(* CODESYS project bibliothek.library
   Company: Viessmann
   Title: GWP_Libary_Visu_1
   Placeholder: GWP_Libary_Visu_1
   Version: 0.0.1

Project tree, tasks and I/O mapping:
  libraries: GWP Library, 17.9.1 (Viessmann); Tc2_Standard, * (Beckhoff Automation GmbH); Tc2_System, * (Beckhoff Automation GmbH); Tc2_Utilities, * (Beckhoff Automation GmbH); Tc3_Module, * (Beckhoff Automation GmbH); VisuDialogs, * (System)
  DUTs/
    GVLs/
      global variables Globale_Uhr
  POUs/
    Funktionsblock/
    program MAIN [ST]
    program test [FBD]
  Version/
    global variables Global_Version
  VISUs/
    Alarmliste/
      visualisation Alarmliste
    Anlageseite_6/
      visualisation Kaeltekreis6_1
      visualisation Sollwertaenderung_C_6_3
      visualisation Zustandsanzeige
    Hauptmenu_3/
      visualisation Fusszeile_50
      visualisation Hauptmenu
      visualisation Kachel_IBN
      visualisation Kachel_Konfiguration
      visualisation Kachel_Kontakt
      visualisation Kachel_Login
      visualisation Kachel_Sollwerte
      visualisation Kachel_Sprachen
      visualisation Kachel_Uhrzeit_einstellen
      visualisation Kachel_Verlaufsdiagramm
      visualisation Kontaktseite
      visualisation Uhr_einstellen
    Heizkurven/
      visualisation Heizkurve
    Home/
      visualisation Auswahlmenue
      visualisation Ein_Aus_Schalter
      visualisation Home_Standard_50
      visualisation RI_Schema_50
    IBN/
      visualisation IO_Auswahl
      visualisation Liste_AI
      visualisation Liste_AO
      visualisation Liste_DI
      visualisation Liste_DO
      visualisation SW_IBN_Einstellungen_K
    Infoseite/
      visualisation Infoliste
      visualisation Infoseite
    Sollwertmenu_9/
      Sollwerte Einstellungen/
        visualisation SW_Einstellungen_C
        visualisation SW_Einstellungen_Faktor
        visualisation SW_Einstellungen_K
        visualisation SW_Einstellungen_min
        visualisation SW_Einstellungen_ms
        visualisation SW_zuruecksetzen
      Sollwertmenu/
        visualisation Sollwertmenu
      Wärmegewinnung/
        UWP/
          visualisation SW_WG_UWP_Verd
          visualisation SW_WG_UWP_Verd_Liste
        visualisation Kachel_Abtauspeicher
        visualisation Kachel_Abtauungen
        visualisation Kachel_Abwaerme
        visualisation Kachel_Erdsonden
        visualisation Kachel_Grundwasser
        visualisation Kachel_Luft
        visualisation Kachel_Tiefhaltung
        visualisation Kachel_UWP_Verd
        visualisation Sollwertmenu_Waermegewinnung
      Wärmepumpe/
        EEV/
          visualisation SW_WP_EEV
          visualisation SW_WP_EEV_Liste
        Einsatzgrenzen/
          visualisation SW_WP_Einsatzgrenzen
          visualisation SW_WP_Einsatzgrenzen_Liste
        visualisation Kachel_Allgemein
        visualisation Kachel_EEV
        visualisation Kachel_Einsatzgrenzen
        visualisation Kachel_Verdichter
        visualisation Sollwertmenu_Waermepumpe
      Wärmesenke/
        visualisation Kachel_Heizgruppen
        visualisation Kachel_Hochhaltung
        visualisation Kachel_HWP
        visualisation Kachel_TWW
        visualisation Kachel_UWP_Verfl
        visualisation Sollwertmenu_Waermesenke
    Sprache/
      visualisation Spracheistellungen
    Zeitprogramm/
      visualisation EIn_Aus_Zeit_aendern
      visualisation Wochenuhr_W7
      visualisation Wochenuhr_W7_Liste
    image pool Icon
    text list Sprachen
    visualisation test_1
  00000000-0000-0000-0000-000000000000|C:\Users\kuzr\Documents\Visual Studio 2013\Bildersammlung_VI\IC_102000\energietraeger_biomasse_fehler.png
  00000000-0000-0000-0000-000000000000|C:\Users\kuzr\Documents\Visual Studio 2013\Bildersammlung_VI\IC_102000\energietraeger_biomasse_inaktiv.png
  00000000-0000-0000-0000-000000000000|C:\Users\kuzr\Documents\Visual Studio 2013\Bildersammlung_VI\IC_102000\energietraeger_gas.png
  00000000-0000-0000-0000-000000000000|C:\Users\kuzr\Documents\Visual Studio 2013\Bildersammlung_VI\IC_102000\energietraeger_gas_fehler.png
  00000000-0000-0000-0000-000000000000|C:\Users\kuzr\Documents\Visual Studio 2013\Bildersammlung_VI\IC_102000\energietraeger_naturwaerme.png
  00000000-0000-0000-0000-000000000000|C:\Users\kuzr\Documents\Visual Studio 2013\Bildersammlung_VI\IC_102000\energietraeger_naturwaerme_fehler (2).png
  00000000-0000-0000-0000-000000000000|C:\Users\kuzr\Documents\Visual Studio 2013\Bildersammlung_VI\IC_102000\energietraeger_naturwaerme_fehler.png
  00000000-0000-0000-0000-000000000000|C:\Users\kuzr\Documents\Visual Studio 2013\Bildersammlung_VI\IC_102000\energietraeger_naturwaerme_inaktiv.png
  00000000-0000-0000-0000-000000000000|C:\Users\kuzr\Documents\Visual Studio 2013\Bildersammlung_VI\IC_102000\energietraeger_oel.png
  00000000-0000-0000-0000-000000000000|C:\Users\kuzr\Documents\Visual Studio 2013\Bildersammlung_VI\IC_102000\energietraeger_oel_inaktiv.png
  00000000-0000-0000-0000-000000000000|C:\Users\kuzr\Documents\Visual Studio 2013\Bildersammlung_VI\IC_102000\heizkreis_direkt (2).png
  00000000-0000-0000-0000-000000000000|C:\Users\kuzr\Documents\Visual Studio 2013\Bildersammlung_VI\IC_102000\heizkreis_direkt.png
  00000000-0000-0000-0000-000000000000|C:\Users\kuzr\Documents\Visual Studio 2013\Bildersammlung_VI\IC_102000\heizkreis_direkt_fehler.png
  00000000-0000-0000-0000-000000000000|C:\Users\kuzr\Documents\Visual Studio 2013\Bildersammlung_VI\IC_102000\heizkreis_direkt_inaktiv (2).png
  00000000-0000-0000-0000-000000000000|C:\Users\kuzr\Documents\Visual Studio 2013\Bildersammlung_VI\IC_102000\heizkreis_direkt_inaktiv.png
  00000000-0000-0000-0000-000000000000|C:\Users\kuzr\Documents\Visual Studio 2013\Bildersammlung_VI\IC_102000\heizkreis_fussbodenheizung.png
  00000000-0000-0000-0000-000000000000|C:\Users\kuzr\Documents\Visual Studio 2013\Bildersammlung_VI\IC_102000\heizkreis_fussbodenheizung_fehler.png
  00000000-0000-0000-0000-000000000000|C:\Users\kuzr\Documents\Visual Studio 2013\Bildersammlung_VI\IC_102000\heizkreis_fussbodenheizung_inaktiv.png
  00000000-0000-0000-0000-000000000000|C:\Users\kuzr\Documents\Visual Studio 2013\Bildersammlung_VI\IC_102000\heizkreis_mischer.png
  00000000-0000-0000-0000-000000000000|C:\Users\kuzr\Documents\Visual Studio 2013\Bildersammlung_VI\IC_102000\heizkreis_mischer_fehler.png
  00000000-0000-0000-0000-000000000000|C:\Users\kuzr\Documents\Visual Studio 2013\Bildersammlung_VI\IC_102000\heizkreis_mischer_inaktiv.png
  00000000-0000-0000-0000-000000000000|C:\Users\kuzr\Documents\Visual Studio 2013\Bildersammlung_VI\IC_102000\IC_102015_klappen_02.png
  00000000-0000-0000-0000-000000000000|C:\Users\kuzr\Documents\Visual Studio 2013\Bildersammlung_VI\IC_102000\klappen_01 (2).png
  00000000-0000-0000-0000-000000000000|C:\Users\kuzr\Documents\Visual Studio 2013\Bildersammlung_VI\IC_102000\klappen_01.png
  00000000-0000-0000-0000-000000000000|C:\Users\kuzr\Documents\Visual Studio 2013\Bildersammlung_VI\IC_102000\klappen_02.png
  00000000-0000-0000-0000-000000000000|C:\Users\kuzr\Documents\Visual Studio 2013\Bildersammlung_VI\IC_102000\komponente_detail_heizkreis.png
  00000000-0000-0000-0000-000000000000|C:\Users\kuzr\Documents\Visual Studio 2013\Bildersammlung_VI\IC_102000\komponente_detail_klappe (2).png
  00000000-0000-0000-0000-000000000000|C:\Users\kuzr\Documents\Visual Studio 2013\Bildersammlung_VI\IC_102000\komponente_detail_klappe.png
  00000000-0000-0000-0000-000000000000|C:\Users\kuzr\Documents\Visual Studio 2013\Bildersammlung_VI\IC_102000\komponente_detail_klappe_fehler (2).png
  00000000-0000-0000-0000-000000000000|C:\Users\kuzr\Documents\Visual Studio 2013\Bildersammlung_VI\IC_102000\komponente_detail_klappe_fehler.png
  00000000-0000-0000-0000-000000000000|C:\Users\kuzr\Documents\Visual Studio 2013\Bildersammlung_VI\IC_102000\komponente_detail_klappe_inaktiv.png
  00000000-0000-0000-0000-000000000000|C:\Users\kuzr\Documents\Visual Studio 2013\Bildersammlung_VI\IC_102000\komponente_detail_klappe_inaktiv_2.png
  00000000-0000-0000-0000-000000000000|C:\Users\kuzr\Documents\Visual Studio 2013\Bildersammlung_VI\IC_102000\komponente_detail_mischer_01.png
  00000000-0000-0000-0000-000000000000|C:\Users\kuzr\Documents\Visual Studio 2013\Bildersammlung_VI\IC_102000\komponente_detail_mischer_02.png
  00000000-0000-0000-0000-000000000000|C:\Users\kuzr\Documents\Visual Studio 2013\Bildersammlung_VI\IC_102000\komponente_detail_mischer_fehler.png
  00000000-0000-0000-0000-000000000000|C:\Users\kuzr\Documents\Visual Studio 2013\Bildersammlung_VI\IC_102000\komponente_detail_mischer_inaktiv.png
  00000000-0000-0000-0000-000000000000|C:\Users\kuzr\Documents\Visual Studio 2013\Bildersammlung_VI\IC_102000\komponente_detail_pumpe.png
  00000000-0000-0000-0000-000000000000|C:\Users\kuzr\Documents\Visual Studio 2013\Bildersammlung_VI\IC_102000\komponente_detail_pumpe_fehler.png
  00000000-0000-0000-0000-000000000000|C:\Users\kuzr\Documents\Visual Studio 2013\Bildersammlung_VI\IC_102000\komponente_detail_pumpe_inaktiv.png
  00000000-0000-0000-0000-000000000000|C:\Users\kuzr\Documents\Visual Studio 2013\Bildersammlung_VI\IC_102000\mischer_01.png
  00000000-0000-0000-0000-000000000000|C:\Users\kuzr\Documents\Visual Studio 2013\Bildersammlung_VI\IC_102000\mischer_02.png
  00000000-0000-0000-0000-000000000000|C:\Users\kuzr\Documents\Visual Studio 2013\Bildersammlung_VI\IC_102000\mischer_03.png
  00000000-0000-0000-0000-000000000000|C:\Users\kuzr\Documents\Visual Studio 2013\Bildersammlung_VI\IC_102000\mischer_04.png
  00000000-0000-0000-0000-000000000000|C:\Users\kuzr\Documents\Visual Studio 2013\Bildersammlung_VI\IC_102000\mischer_05.png
  00000000-0000-0000-0000-000000000000|C:\Users\kuzr\Documents\Visual Studio 2013\Bildersammlung_VI\IC_102000\mischer_06.png
  00000000-0000-0000-0000-000000000000|C:\Users\kuzr\Documents\Visual Studio 2013\Bildersammlung_VI\IC_102000\mischer_07.png
  00000000-0000-0000-0000-000000000000|C:\Users\kuzr\Documents\Visual Studio 2013\Bildersammlung_VI\IC_102000\mischer_08.png
  00000000-0000-0000-0000-000000000000|C:\Users\kuzr\Documents\Visual Studio 2013\Bildersammlung_VI\IC_102000\mischer_09.png
  00000000-0000-0000-0000-000000000000|C:\Users\kuzr\Documents\Visual Studio 2013\Bildersammlung_VI\IC_102000\mischer_10.png
  00000000-0000-0000-0000-000000000000|C:\Users\kuzr\Documents\Visual Studio 2013\Bildersammlung_VI\IC_102000\mischer_11.png
  00000000-0000-0000-0000-000000000000|C:\Users\kuzr\Documents\Visual Studio 2013\Bildersammlung_VI\IC_102000\mischer_12.png
  00000000-0000-0000-0000-000000000000|C:\Users\kuzr\Documents\Visual Studio 2013\Bildersammlung_VI\IC_102000\pumpe_links.png
  00000000-0000-0000-0000-000000000000|C:\Users\kuzr\Documents\Visual Studio 2013\Bildersammlung_VI\IC_102000\pumpe_oben.png
  00000000-0000-0000-0000-000000000000|C:\Users\kuzr\Documents\Visual Studio 2013\Bildersammlung_VI\IC_102000\pumpe_rechts.png
  00000000-0000-0000-0000-000000000000|C:\Users\kuzr\Documents\Visual Studio 2013\Bildersammlung_VI\IC_102000\pumpe_unten.png
  00000000-0000-0000-0000-000000000000|C:\Users\kuzr\Documents\Visual Studio 2013\Bildersammlung_VI\IC_102000\speicher_eis.png
  00000000-0000-0000-0000-000000000000|C:\Users\kuzr\Documents\Visual Studio 2013\Bildersammlung_VI\IC_102000\speicher_eis_fehler.png
  00000000-0000-0000-0000-000000000000|C:\Users\kuzr\Documents\Visual Studio 2013\Bildersammlung_VI\IC_102000\speicher_eis_inaktiv.png
  00000000-0000-0000-0000-000000000000|C:\Users\kuzr\Documents\Visual Studio 2013\Bildersammlung_VI\IC_102000\speicher_heizen.png
  00000000-0000-0000-0000-000000000000|C:\Users\kuzr\Documents\Visual Studio 2013\Bildersammlung_VI\IC_102000\speicher_heizen_fehler.png
  00000000-0000-0000-0000-000000000000|C:\Users\kuzr\Documents\Visual Studio 2013\Bildersammlung_VI\IC_102000\speicher_heizen_inaktiv.png
  00000000-0000-0000-0000-000000000000|C:\Users\kuzr\Documents\Visual Studio 2013\Bildersammlung_VI\IC_102000\speicher_warmwasser.png
  00000000-0000-0000-0000-000000000000|C:\Users\kuzr\Documents\Visual Studio 2013\Bildersammlung_VI\IC_102000\speicher_warmwasser_fehler.png
  00000000-0000-0000-0000-000000000000|C:\Users\kuzr\Documents\Visual Studio 2013\Bildersammlung_VI\IC_102000\speicher_warmwasser_inaktiv.png
  00000000-0000-0000-0000-000000000000|C:\Users\kuzr\Documents\Visual Studio 2013\Bildersammlung_VI\IC_102000\energietraeger_biomasse.png
  00000000-0000-0000-0000-000000000000|C:\Users\kuzr\Documents\Visual Studio 2013\Bildersammlung_VI\IC_106000\komponente_brenner.png
  00000000-0000-0000-0000-000000000000|C:\Users\kuzr\Documents\Visual Studio 2013\Bildersammlung_VI\IC_106000\komponente_brenner_fehler.png
  00000000-0000-0000-0000-000000000000|C:\Users\kuzr\Documents\Visual Studio 2013\Bildersammlung_VI\IC_106000\komponente_brenner_inaktiv.png
  00000000-0000-0000-0000-000000000000|C:\Users\kuzr\Documents\Visual Studio 2013\Bildersammlung_VI\IC_106000\speicher.png
  00000000-0000-0000-0000-000000000000|C:\Users\kuzr\Documents\Visual Studio 2013\Bildersammlung_VI\IC_106000\speicher_eis.png
  00000000-0000-0000-0000-000000000000|C:\Users\kuzr\Documents\Visual Studio 2013\Bildersammlung_VI\IC_106000\system_leistung_nicht_touchbar.png
  00000000-0000-0000-0000-000000000000|C:\Users\kuzr\Documents\Visual Studio 2013\Bildersammlung_VI\IC_106000\system_leistung_touchbar.png
  00000000-0000-0000-0000-000000000000|C:\Users\kuzr\Documents\Visual Studio 2013\Bildersammlung_VI\IC_106000\waermetauscher.png
  00000000-0000-0000-0000-000000000000|C:\Users\kuzr\Documents\Visual Studio 2013\Bildersammlung_VI\IC_106000\weiche.png
  00000000-0000-0000-0000-000000000000|C:\Users\kuzr\Documents\Visual Studio 2013\Bildersammlung_VI\IC_108000\komponente_brenner_fehler.png
  00000000-0000-0000-0000-000000000000|C:\Users\kuzr\Documents\Visual Studio 2013\Bildersammlung_VI\IC_108000\komponente_brenner_inaktiv.png
  00000000-0000-0000-0000-000000000000|C:\Users\kuzr\Documents\Visual Studio 2013\Bildersammlung_VI\IC_108000\speicher.png
  00000000-0000-0000-0000-000000000000|C:\Users\kuzr\Documents\Visual Studio 2013\Bildersammlung_VI\IC_108000\speicher_eis.png
  00000000-0000-0000-0000-000000000000|C:\Users\kuzr\Documents\Visual Studio 2013\Bildersammlung_VI\IC_108000\komponente_brenner.png
  00000000-0000-0000-0000-000000000000|C:\Users\kuzr\Documents\Visual Studio 2013\Bildersammlung_VI\IC_111000\bildschirm_reinigen.png
  00000000-0000-0000-0000-000000000000|C:\Users\kuzr\Documents\Visual Studio 2013\Bildersammlung_VI\IC_111000\dokumentation.png
  00000000-0000-0000-0000-000000000000|C:\Users\kuzr\Documents\Visual Studio 2013\Bildersammlung_VI\IC_111000\kontaktdaten_nutzer.png
  00000000-0000-0000-0000-000000000000|C:\Users\kuzr\Documents\Visual Studio 2013\Bildersammlung_VI\IC_111000\kontaktdaten_viessmann.png
  00000000-0000-0000-0000-000000000000|C:\Users\kuzr\Documents\Visual Studio 2013\Bildersammlung_VI\IC_111000\nutzeranmeldung.png
  00000000-0000-0000-0000-000000000000|C:\Users\kuzr\Documents\Visual Studio 2013\Bildersammlung_VI\IC_111000\oberflaeche_schließen.png
  00000000-0000-0000-0000-000000000000|C:\Users\kuzr\Documents\Visual Studio 2013\Bildersammlung_VI\IC_111000\pruefbetrieb.png
  00000000-0000-0000-0000-000000000000|C:\Users\kuzr\Documents\Visual Studio 2013\Bildersammlung_VI\IC_111000\system_konfigurieren.png
  00000000-0000-0000-0000-000000000000|C:\Users\kuzr\Documents\Visual Studio 2013\Bildersammlung_VI\IC_111000\betriebszaehler_zuruecksetzen.png
  00000000-0000-0000-0000-000000000000|C:\Users\kuzr\Documents\Visual Studio 2013\Bildersammlung_VI\IC_112000\abschaltbetrieb.png
  00000000-0000-0000-0000-000000000000|C:\Users\kuzr\Documents\Visual Studio 2013\Bildersammlung_VI\IC_112000\aktiv.png
  00000000-0000-0000-0000-000000000000|C:\Users\kuzr\Documents\Visual Studio 2013\Bildersammlung_VI\IC_112000\an.png
  00000000-0000-0000-0000-000000000000|C:\Users\kuzr\Documents\Visual Studio 2013\Bildersammlung_VI\IC_112000\astatur_01.png
  00000000-0000-0000-0000-000000000000|C:\Users\kuzr\Documents\Visual Studio 2013\Bildersammlung_VI\IC_112000\auf.png
  00000000-0000-0000-0000-000000000000|C:\Users\kuzr\Documents\Visual Studio 2013\Bildersammlung_VI\IC_112000\aus.png
  00000000-0000-0000-0000-000000000000|C:\Users\kuzr\Documents\Visual Studio 2013\Bildersammlung_VI\IC_112000\bedingung_erfuellt.png
  00000000-0000-0000-0000-000000000000|C:\Users\kuzr\Documents\Visual Studio 2013\Bildersammlung_VI\IC_112000\bedingung_nicht_erfuellt.png
  00000000-0000-0000-0000-000000000000|C:\Users\kuzr\Documents\Visual Studio 2013\Bildersammlung_VI\IC_112000\email_prueftaste.png
  00000000-0000-0000-0000-000000000000|C:\Users\kuzr\Documents\Visual Studio 2013\Bildersammlung_VI\IC_112000\erfuellt.png
  00000000-0000-0000-0000-000000000000|C:\Users\kuzr\Documents\Visual Studio 2013\Bildersammlung_VI\IC_112000\exportieren.png
  00000000-0000-0000-0000-000000000000|C:\Users\kuzr\Documents\Visual Studio 2013\Bildersammlung_VI\IC_112000\frostschutzbetrieb.png
  00000000-0000-0000-0000-000000000000|C:\Users\kuzr\Documents\Visual Studio 2013\Bildersammlung_VI\IC_112000\haeckchen_ungesetzt (2).png
  00000000-0000-0000-0000-000000000000|C:\Users\kuzr\Documents\Visual Studio 2013\Bildersammlung_VI\IC_112000\haeckchen_ungesetzt.png
  00000000-0000-0000-0000-000000000000|C:\Users\kuzr\Documents\Visual Studio 2013\Bildersammlung_VI\IC_112000\home.png
  00000000-0000-0000-0000-000000000000|C:\Users\kuzr\Documents\Visual Studio 2013\Bildersammlung_VI\IC_112000\home_uebersicht.png
  00000000-0000-0000-0000-000000000000|C:\Users\kuzr\Documents\Visual Studio 2013\Bildersammlung_VI\IC_112000\inaktiv.png
  00000000-0000-0000-0000-000000000000|C:\Users\kuzr\Documents\Visual Studio 2013\Bildersammlung_VI\IC_112000\intervall.png
  00000000-0000-0000-0000-000000000000|C:\Users\kuzr\Documents\Visual Studio 2013\Bildersammlung_VI\IC_112000\Itastatur_03.png
  00000000-0000-0000-0000-000000000000|C:\Users\kuzr\Documents\Visual Studio 2013\Bildersammlung_VI\IC_112000\ja.png
  00000000-0000-0000-0000-000000000000|C:\Users\kuzr\Documents\Visual Studio 2013\Bildersammlung_VI\IC_112000\kopieren.png
  00000000-0000-0000-0000-000000000000|C:\Users\kuzr\Documents\Visual Studio 2013\Bildersammlung_VI\IC_112000\laden.png
  00000000-0000-0000-0000-000000000000|C:\Users\kuzr\Documents\Visual Studio 2013\Bildersammlung_VI\IC_112000\listenansicht.png
  00000000-0000-0000-0000-000000000000|C:\Users\kuzr\Documents\Visual Studio 2013\Bildersammlung_VI\IC_112000\meldelisten_archiv.png
  00000000-0000-0000-0000-000000000000|C:\Users\kuzr\Documents\Visual Studio 2013\Bildersammlung_VI\IC_112000\meldelisten_einstellungen.png
  00000000-0000-0000-0000-000000000000|C:\Users\kuzr\Documents\Visual Studio 2013\Bildersammlung_VI\IC_112000\meldungen_weiterleiten.png
  00000000-0000-0000-0000-000000000000|C:\Users\kuzr\Documents\Visual Studio 2013\Bildersammlung_VI\IC_112000\menue.png
  00000000-0000-0000-0000-000000000000|C:\Users\kuzr\Documents\Visual Studio 2013\Bildersammlung_VI\IC_112000\minus.png
  00000000-0000-0000-0000-000000000000|C:\Users\kuzr\Documents\Visual Studio 2013\Bildersammlung_VI\IC_112000\nein.png
  00000000-0000-0000-0000-000000000000|C:\Users\kuzr\Documents\Visual Studio 2013\Bildersammlung_VI\IC_112000\nicht_erfuellt.png
  00000000-0000-0000-0000-000000000000|C:\Users\kuzr\Documents\Visual Studio 2013\Bildersammlung_VI\IC_112000\normalbetrieb.png
  00000000-0000-0000-0000-000000000000|C:\Users\kuzr\Documents\Visual Studio 2013\Bildersammlung_VI\IC_112000\pfeil_rechts.png
  00000000-0000-0000-0000-000000000000|C:\Users\kuzr\Documents\Visual Studio 2013\Bildersammlung_VI\IC_112000\plus.png
  00000000-0000-0000-0000-000000000000|C:\Users\kuzr\Documents\Visual Studio 2013\Bildersammlung_VI\IC_112000\quittieren_aus.png
  00000000-0000-0000-0000-000000000000|C:\Users\kuzr\Documents\Visual Studio 2013\Bildersammlung_VI\IC_112000\quittierena_an.png
  00000000-0000-0000-0000-000000000000|C:\Users\kuzr\Documents\Visual Studio 2013\Bildersammlung_VI\IC_112000\radiobutton_gesetzt.png
  00000000-0000-0000-0000-000000000000|C:\Users\kuzr\Documents\Visual Studio 2013\Bildersammlung_VI\IC_112000\radiobutton_ungesetzt.png
  text list GlobalTextList
*)

// DUTs/GVLs/Globale_Uhr
{attribute 'qualified_only'}
VAR_GLOBAL
	
	   systemtimestruct		: timestruct;   
END_VAR

// Version/Global_Version
{attribute 'TcGenerated'}
// This function has been automatically generated from the project information.
VAR_GLOBAL CONSTANT
	{attribute 'const_non_replaced'}
	{attribute 'linkalways'}
	stLibVersion_GWP_Libary_Visu_1 : ST_LibVersion := (iMajor := 0, iMinor := 0, iBuild := 1, iRevision := 0, sVersion := '0.0.1');
END_VAR

// POUs/MAIN
PROGRAM MAIN
VAR

	

END_VAR

END_PROGRAM

// POUs/test
PROGRAM test
VAR

	
	Globale_Zeit_0: Globale_Zeit;
    CLK_W_0: CLK_W;
	
	GR_2_0: GR_2;
	
	


	
	Logger_0: Logger;
	GR_4_mit_RE_0: GR_4_mit_RE;
	CLK_W7_0: CLK_W7;
END_VAR

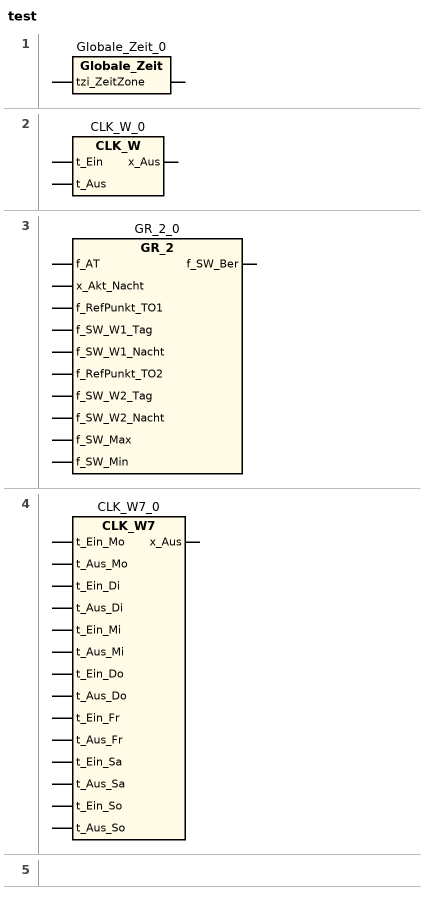
// NETWORK 1
Globale_Zeit_0(); // Globale_Zeit

// NETWORK 2
CLK_W_0(); // CLK_W

// NETWORK 3
GR_2_0(); // GR_2

// NETWORK 4
CLK_W7_0(); // CLK_W7

// NETWORK 5

END_PROGRAM

// VISUs/Alarmliste/Alarmliste
VISUALIZATION Alarmliste  // 800x430
END_VISUALIZATION

// VISUs/Anlageseite_6/Kaeltekreis6_1
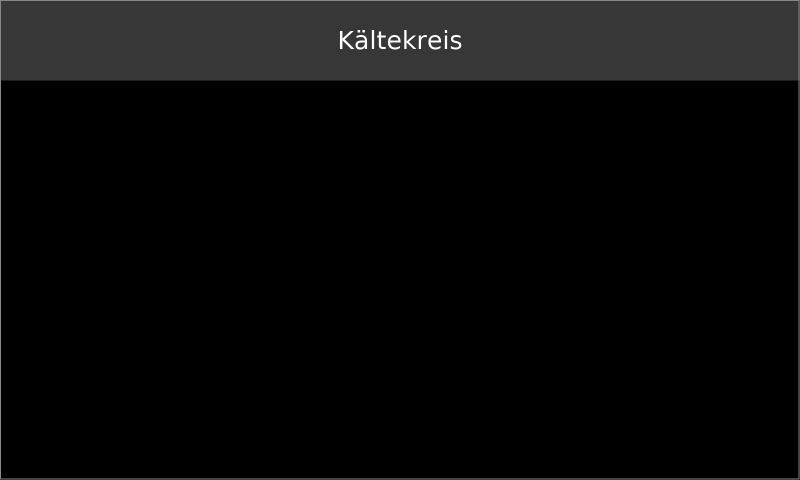
VISUALIZATION Kaeltekreis6_1  // 800x480
    Rectangle (0,0 800x80), "Kältekreis"
END_VISUALIZATION

// VISUs/Anlageseite_6/Sollwertaenderung_C_6_3
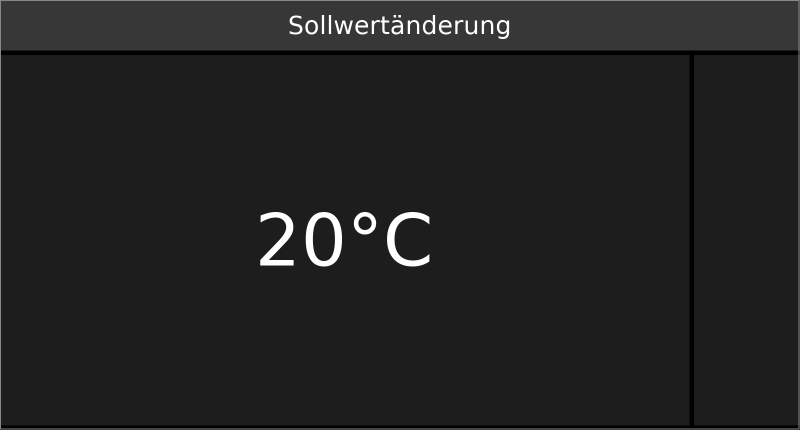
VISUALIZATION Sollwertaenderung_C_6_3  // 800x430
    Rectangle (0,0 800x50), "Sollwertänderung"
    Rectangle (0,55 689x370), "20°C"
    Rectangle (694,55 106x370)
END_VISUALIZATION

// VISUs/Anlageseite_6/Zustandsanzeige
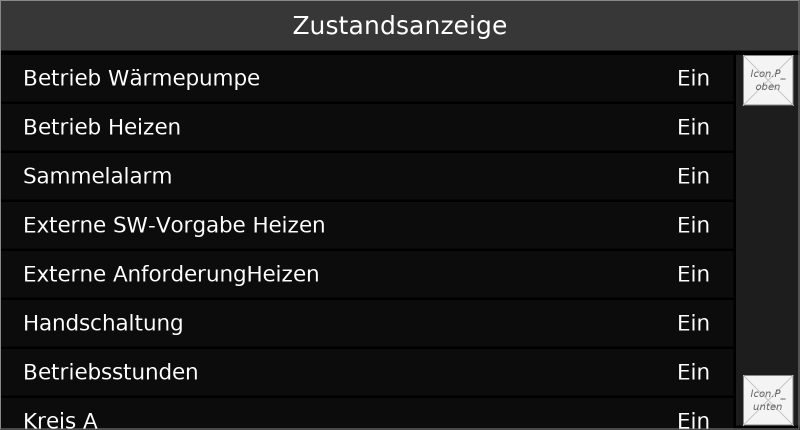
VISUALIZATION Zustandsanzeige  // 800x430
VAR_IN_OUT
	auf:BOOL;
		
END_VAR
    Image (1113,281 30x116), image: Icon.waermetauscher
    Group (0,0 800x640)
        Rectangle (0,0 800x50), "Zustandsanzeige"
        Group (0,430 800x50)
            Rectangle (0,0 800x50)
            Image (25,0 50x50), image: Icon.home
            Image (425,0 50x50), image: Icon.reinnavigieren
            Image (625,0 50x50), image: Icon.warnung_rot
            Image (125,0 50x50), image: Icon.zurueck
            Image (325,0 50x50), image: Icon.reinnavigieren
            Image (325,0 50x50), image: Icon.p_links
            Image (425,0 50x50), image: Icon.P_rechts
        Rectangle (0,55 733x46)
        Label (20,55 479x46), "Betrieb Wärmepumpe"
        Rectangle (0,104 733x46)
        Label (20,104 479x46), "Betrieb Heizen"
        Rectangle (0,153 733x46)
        Label (20,153 479x46), "Sammelalarm"
        Rectangle (0,202 733x46)
        Label (20,202 479x46), "Externe SW-Vorgabe Heizen"
        Rectangle (0,251 733x46)
        Label (20,251 479x46), "Externe AnforderungHeizen"
        Rectangle (0,300 733x46)
        Label (20,300 479x46), "Handschaltung"
        Rectangle (0,349 733x46)
        Label (20,349 479x46), "Betriebsstunden"
        Rectangle (583,55 130x46), "Ein"
        Rectangle (583,104 130x46), "Ein"
        Rectangle (0,398 733x46)
        Label (20,398 479x46), "Kreis A"
        Rectangle (0,447 733x46)
        Label (20,447 479x46), "Kreis B"
        Rectangle (0,496 733x46)
        Label (20,496 479x46), "Stufe 1"
        Rectangle (0,545 733x46)
        Label (20,545 479x46), "Stufe 2"
        Rectangle (583,545 130x46), "Ein"
        Rectangle (0,594 733x46)
        Label (20,594 479x46), "Stufe 3"
        Rectangle (583,153 130x46), "Ein"
        Rectangle (583,202 130x46), "Ein"
        Rectangle (583,251 130x46), "Ein"
        Rectangle (583,349 130x46), "Ein"
        Rectangle (583,300 130x46), "Ein"
        Rectangle (583,398 130x46), "Ein"
        Rectangle (583,447 130x46), "Ein"
        Rectangle (583,496 130x46), "Ein"
        Rectangle (583,594 130x46), "Ein"
        Rectangle (736,55 64x370)
        Image (743,55 50x50), image: Icon.P_oben
            OnMouseClick: write the text variable via Default
        Image (743,375 50x50), image: Icon.P_unten
END_VISUALIZATION

// VISUs/Hauptmenu_3/Fusszeile_50
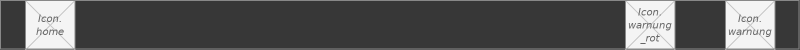
VISUALIZATION Fusszeile_50  // 800x50
    Group (0,0 800x50)
        Rectangle (0,0 800x50)
        Image (625,0 50x50), image: Icon.warnung_rot
            OnMouseClick: execute { GWP_Library.Visu.i_Frame_Index:=0; }
        Image (25,0 50x50), image: Icon.home
            OnMouseClick:  Assign=Home_Standard_50, Type=Assignment
            OnMouseClick: execute { GWP_Library.Visu.i_Frame_Index:=0; }
        Image (725,0 50x50), image: Icon.warnung
            OnMouseClick:  Assign=Infoseite, Type=Assignment
            OnMouseClick: execute { GWP_Library.Visu.i_Frame_Index:=0; }
END_VISUALIZATION

// VISUs/Hauptmenu_3/Hauptmenu
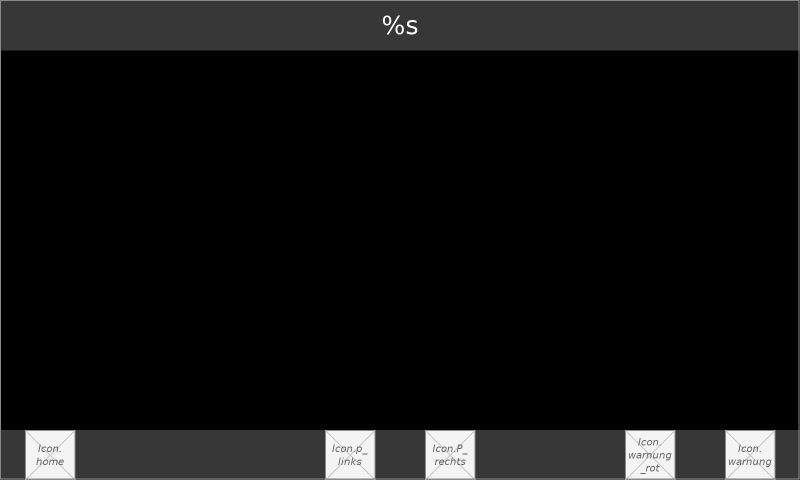
VISUALIZATION Hauptmenu  // 800x480
VAR_IN_OUT
		
END_VAR

VAR
	i_verschieben:INT;

END_VAR
    Image (425,430 50x50), image: Icon.reinnavigieren
    Image (325,430 50x50), image: Icon.reinnavigieren
    Rectangle (0,0 800x50), "%s", text list: 'Sprachen', text index: 32
    Frame (0,430 800x50)
        shows Fusszeile_50()
    Image (425,430 50x50), image: Icon.P_rechts
        OnMouseClick: execute {
            IF i_verschieben>-800 THEN
            	i_verschieben:=i_verschieben-800;
            END_IF
        }
    Image (325,430 50x50), image: Icon.p_links
        OnMouseClick: execute {
            IF i_verschieben<0 THEN
            	i_verschieben:=i_verschieben+800;
            END_IF
        }
    Rectangle (88,515 454x57), "Kachel 1: 0;55 *** Kachel 2: 201;55 *** Kachel 3: 402;55 *** Kachel 4: 604;55 Kachel 5: 0;242 *** Kachel 6: 201;242 *** Kachel 7: 402;242 *** Kachel 8: 604;242"
END_VISUALIZATION

// VISUs/Hauptmenu_3/Kachel_IBN
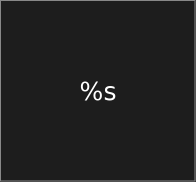
VISUALIZATION Kachel_IBN  // 196x182
    Rectangle (0,0 196x182), "%s", text list: 'Sprachen', text index: 38
END_VISUALIZATION

// VISUs/Hauptmenu_3/Kachel_Konfiguration
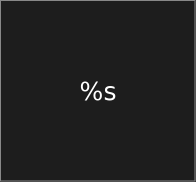
VISUALIZATION Kachel_Konfiguration  // 196x182
    Rectangle (0,0 196x182), "%s", text list: 'Sprachen', text index: 39
END_VISUALIZATION

// VISUs/Hauptmenu_3/Kachel_Kontakt
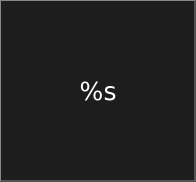
VISUALIZATION Kachel_Kontakt  // 196x182
    Rectangle (0,0 196x182), "%s", text list: 'Sprachen', text index: 40
END_VISUALIZATION

// VISUs/Hauptmenu_3/Kachel_Login
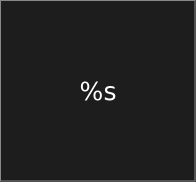
VISUALIZATION Kachel_Login  // 196x182
    Rectangle (0,0 196x182), "%s", text list: 'Sprachen', text index: 34
END_VISUALIZATION

// VISUs/Hauptmenu_3/Kachel_Sollwerte
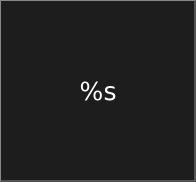
VISUALIZATION Kachel_Sollwerte  // 196x182
    Rectangle (0,0 196x182), "%s", text list: 'Sprachen', text index: 35
END_VISUALIZATION

// VISUs/Hauptmenu_3/Kachel_Sprachen
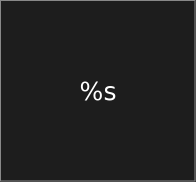
VISUALIZATION Kachel_Sprachen  // 196x182
    Rectangle (0,0 196x182), "%s", text list: 'Sprachen', text index: 33
END_VISUALIZATION

// VISUs/Hauptmenu_3/Kachel_Uhrzeit_einstellen
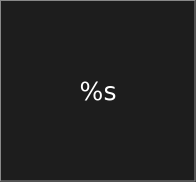
VISUALIZATION Kachel_Uhrzeit_einstellen  // 196x182
    Rectangle (0,0 196x182), "%s", text list: 'Sprachen', text index: 37
END_VISUALIZATION

// VISUs/Hauptmenu_3/Kachel_Verlaufsdiagramm
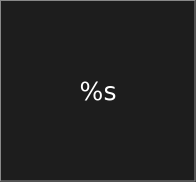
VISUALIZATION Kachel_Verlaufsdiagramm  // 196x182
    Rectangle (0,0 196x182), "%s", text list: 'Sprachen', text index: 36
END_VISUALIZATION

// VISUs/Hauptmenu_3/Kontaktseite
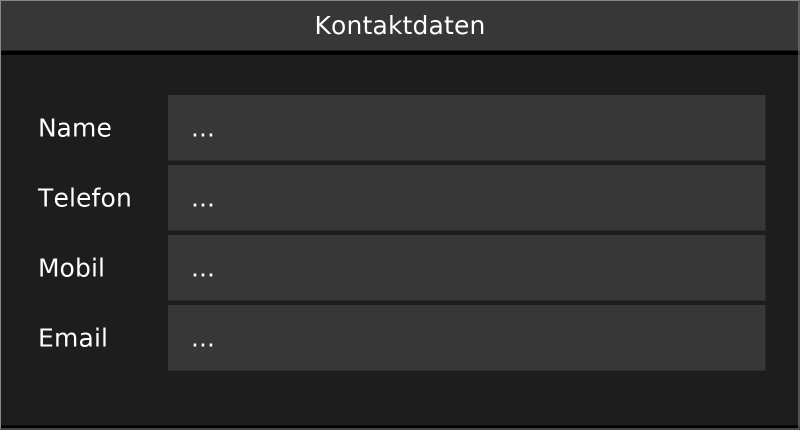
VISUALIZATION Kontaktseite  // 800x430
    Rectangle (0,0 800x50), "Kontaktdaten"
    Rectangle (0,55 800x370)
    Rectangle (168,95 597x65)
    Rectangle (168,165 597x65)
    Rectangle (168,235 597x65)
    Rectangle (168,305 597x65)
    Label (35,95 113x65), "Name"
    Label (35,165 113x65), "Telefon"
    Label (35,235 113x65), "Mobil"
    Label (35,305 113x65), "Email"
    Label (188,305 557x65), "..."
    Label (188,235 557x65), "..."
    Label (188,165 557x65), "..."
    Label (188,95 557x65), "..."
    Frame (0,430 800x50)
        shows Fusszeile_50()
END_VISUALIZATION

// VISUs/Hauptmenu_3/Uhr_einstellen
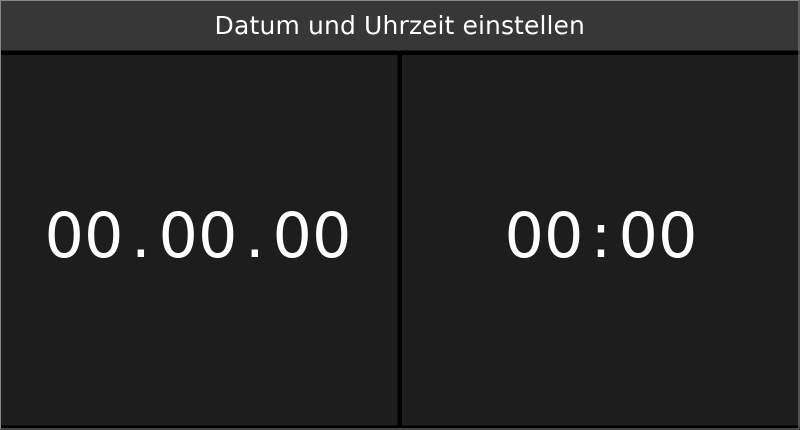
VISUALIZATION Uhr_einstellen  // 800x430
    Frame (0,430 800x50)
        shows Fusszeile_50()
    Rectangle (0,0 800x50), "Datum und Uhrzeit einstellen"
    Rectangle (0,55 397x370)
    Image (425,430 50x50), image: Icon.reinnavigieren
    Image (125,430 50x50), image: Icon.zurueck
        OnMouseClick:  Assign=Hauptmenu, Type=Assignment
    Image (325,430 50x50), image: Icon.reinnavigieren
    Group (402,55 398x370)
        Rectangle (0,0 398x370)
        Group (100,138 198x84)
            Rectangle (84,0 30x84), ":"
            Rectangle (0,0 84x84), "00"
            Rectangle (114,0 84x84), "00"
    Rectangle (156,193 84x84), "00"
    Rectangle (126,193 30x84), "."
    Rectangle (42,193 84x84), "00"
    Rectangle (240,193 30x84), "."
    Rectangle (270,193 84x84), "00"
END_VISUALIZATION

// VISUs/Heizkurven/Heizkurve
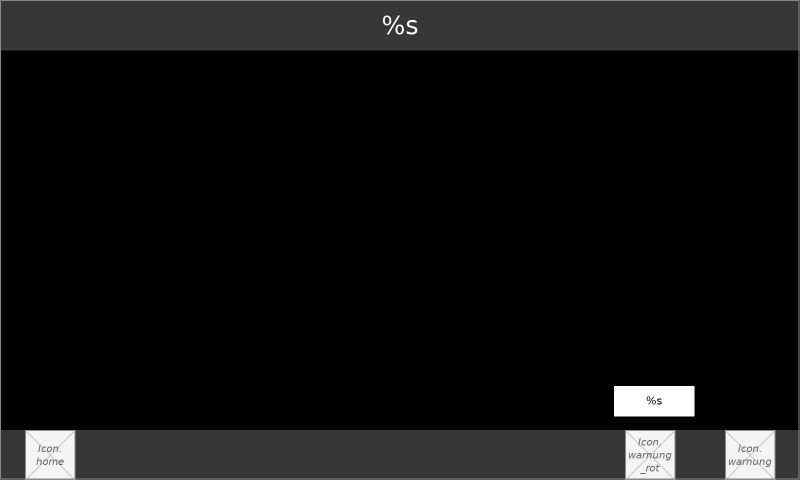
VISUALIZATION Heizkurve  // 800x480
    Image (425,430 50x50), image: Icon.reinnavigieren
    Image (325,430 50x50), image: Icon.reinnavigieren
    Rectangle (0,0 800x50), "%s", text list: 'Sprachen', text index: 71
    Frame (0,430 800x50)
        shows Fusszeile_50()
    Line (154,406)
    Line (143,379) (658,379)
    Line (143,379) (143,90)
    Rectangle (613,385 82x32), "%s"
END_VISUALIZATION

// VISUs/Home/Auswahlmenue
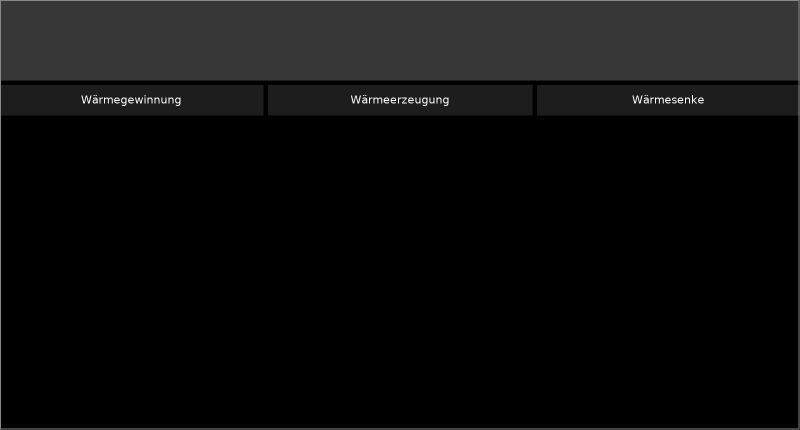
VISUALIZATION Auswahlmenue  // 800x430
    Rectangle (0,0 800x80)
    Rectangle (0,85 263x30), "Wärmegewinnung"
    Rectangle (268,85 264x30), "Wärmeerzeugung"
    Rectangle (537,85 263x30), "Wärmesenke"
END_VISUALIZATION

// VISUs/Home/Ein_Aus_Schalter
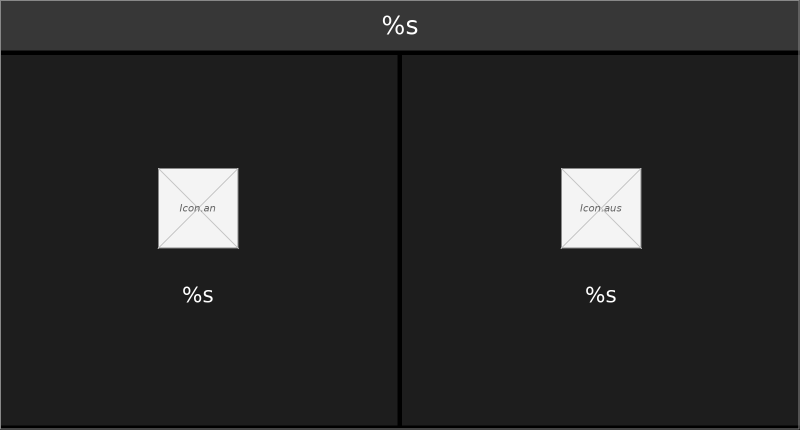
VISUALIZATION Ein_Aus_Schalter  // 800x430
VAR_IN_OUT
	
	i_Status:INT;
END_VAR

VAR_OUTPUT
	

END_VAR

VAR_INPUT
	i_Titel:INT;
	i_Text_1:INT;
	i_Text_2:INT;	

	
END_VAR
    Rectangle (0,0 800x50), "%s", text list: 'Sprachen', text index: i_Titel
    Rectangle (0,55 397x370)
    Rectangle (0,55 397x5)
    Image (158,168 80x80), image: Icon.an
    Rectangle (123,280 150x30), "%s", text list: 'Sprachen', text index: i_Text_1
        OnMouseClick: execute { i_Status:=i_Text_1; }
    Image (125,430 50x50), image: Icon.zurueck
        OnMouseClick: execute { GWP_Library.Visu.i_Frame_Index:=0; }
    Polygon (943,131)
    Rectangle (402,55 398x370)
    Rectangle (402,55 398x5)
    Rectangle (526,280 150x30), "%s", text list: 'Sprachen', text index: i_Text_2
        OnMouseClick: execute { i_Status:=i_Text_2; }
    Image (561,168 80x80), image: Icon.aus
END_VISUALIZATION

// VISUs/Home/Home_Standard_50
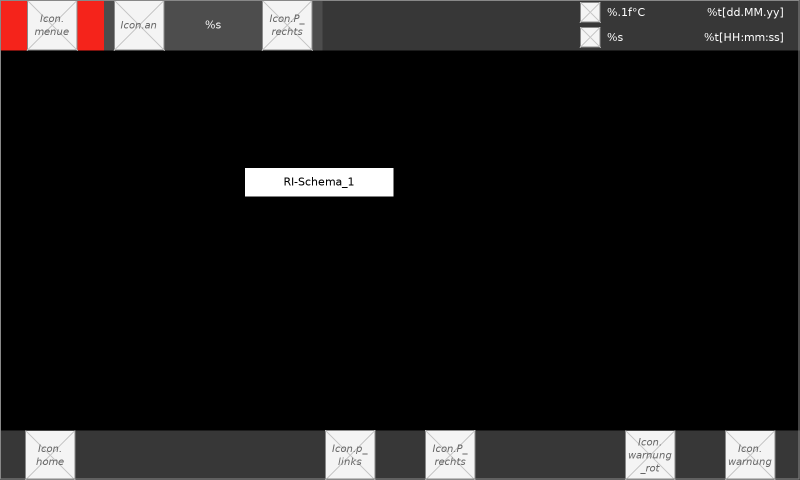
VISUALIZATION Home_Standard_50  // 800x480
VAR_INPUT

END_VAR
	
VAR
	i_Anzeige:INT;	

	

END_VAR
    Frame (0,430 800x50)
        shows Fusszeile_50()
    Frame (0,0 800x430), frame switch variable: GWP_Library.Visu.i_Frame_Index
        shows RI_Schema_50(i_Status := i_Anzeige)
        shows Ein_Aus_Schalter(i_Titel := 41, i_Text_1 := 42, i_Text_2 := 43, i_Status := i_Anzeige)
END_VISUALIZATION

// VISUs/Home/RI_Schema_50
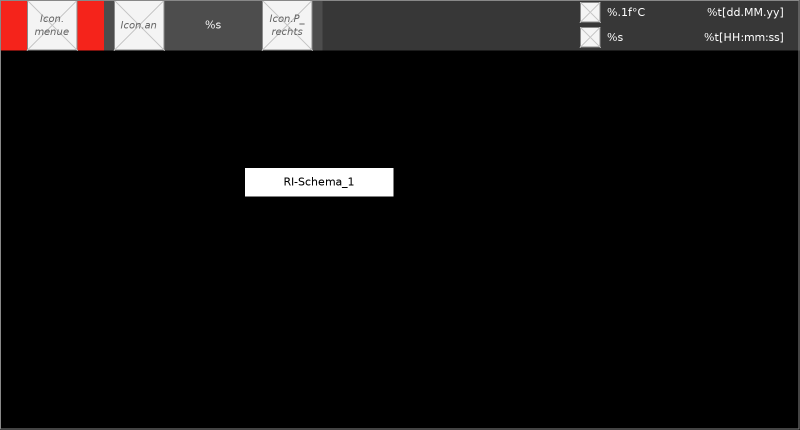
VISUALIZATION RI_Schema_50  // 800x430
VAR
	i_verschieben:INT;
	
END_VAR

VAR_INPUT
	i_Status:INT;

	
	
	
	
END_VAR
    Rectangle (0,0 800x50)
    Rectangle (702,0 85x25), "%t[dd.MM.yy]"
    Rectangle (702,25 85x25), "%t[HH:mm:ss]"
    Image (580,27 20x20), image: Icon.login_status
    Rectangle (604,0 85x25), "%.1f°C"
    Rectangle (604,25 85x25), "%s"
    Group (0,0 104x50)
        OnMouseClick:  Assign=Hauptmenu, Type=Assignment
        Rectangle (0,0 104x50)
        Image (27,0 50x50), image: Icon.menue
    Image (425,430 50x50), image: Icon.P_rechts
        OnMouseClick: execute {
            IF i_verschieben>-800 THEN
            	i_verschieben:=i_verschieben-400;
            END_IF
        }
    Image (325,430 50x50), image: Icon.p_links
        OnMouseClick: execute {
            IF i_verschieben<0 THEN
            	i_verschieben:=i_verschieben+400;
            END_IF
        }
    Image (580,2 20x20), image: Icon.aussentemperatur
    Rectangle (104,0 218x50), "%s", text list: 'Sprachen', text index: i_Status
    Image (114,0 50x50), image: Icon.an
    Image (262,0 50x50), image: Icon.P_rechts
        OnMouseClick: execute { GWP_Library.Visu.i_Frame_Index:=1; }
    Group (244,167 842x88)
        p3560616238: i_verschieben
        Rectangle (0,0 150x30), "RI-Schema_1"
        Rectangle (698,58 150x30), "RI-Schema_2"
END_VISUALIZATION

// VISUs/IBN/IO_Auswahl
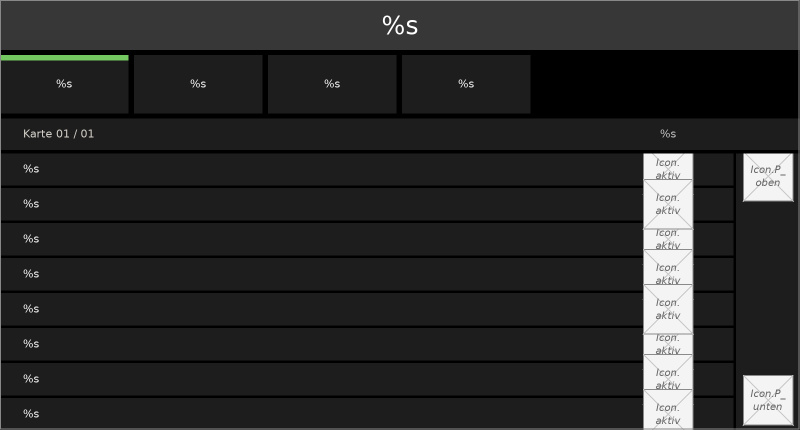
VISUALIZATION IO_Auswahl  // 800x430
    Frame (0,0 800x430), frame switch variable: GWP_Library.Visu.i_Frame_Index
        shows Liste_DI()
        shows Liste_DO()
        shows Liste_AI()
        shows Liste_AO()
        shows SW_IBN_Einstellungen_K(i_titel := 69)
    Frame (0,430 800x50)
        shows Fusszeile_50()
END_VISUALIZATION

// VISUs/IBN/Liste_AI
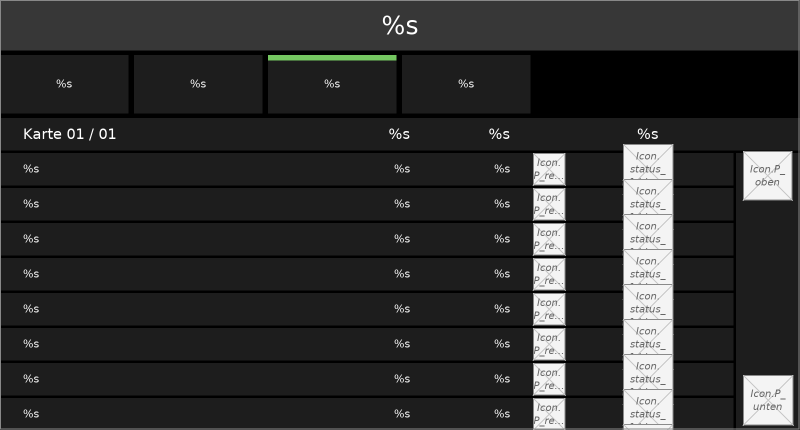
VISUALIZATION Liste_AI  // 800x430
    Rectangle (736,153 64x277)
    Image (743,375 50x50), image: Icon.P_unten
        OnMouseClick: execute {  }
    Image (743,151 49x49), image: Icon.P_oben
    Rectangle (0,153 733x32)
    Rectangle (20,153 400x32), "%s"
    Rectangle (0,223 733x32)
    Rectangle (20,223 400x32), "%s"
    Rectangle (0,188 733x32)
    Rectangle (20,188 400x32), "%s"
    Rectangle (0,258 733x32)
    Rectangle (20,258 400x32), "%s"
    Rectangle (0,328 733x32)
    Rectangle (20,328 400x32), "%s"
    Rectangle (0,293 733x32)
    Rectangle (20,293 400x32), "%s"
    Rectangle (0,538 733x32)
    Rectangle (20,538 400x32), "%s"
    Rectangle (0,363 733x32)
    Rectangle (20,363 400x32), "%s"
    Rectangle (0,433 733x32)
    Rectangle (20,433 400x32), "%s"
    Rectangle (0,398 733x32)
    Rectangle (20,398 400x32), "%s"
    Rectangle (0,468 733x32)
    Rectangle (20,468 400x32), "%s"
    Rectangle (0,503 733x32)
    Rectangle (20,503 400x32), "%s"
    Rectangle (0,118 800x32)
    Rectangle (20,118 324x32), "Karte 01 / 01"
    Rectangle (623,118 50x32), "%s", text list: 'Sprachen', text index: 49
    Image (623,144 50x50), image: Icon.status_fehlerfrei_element
    Image (623,144 50x50), image: Icon.status_fehler_element
    Image (533,153 32x32), image: Icon.P_rechts
        OnMouseClick: execute { GWP_Library.Visu.i_Frame_Index:=4; }
    Rectangle (433,153 80x32), "%s"
    Rectangle (333,153 80x32), "%s"
    Rectangle (433,118 80x32), "%s", text list: 'Sprachen', text index: 50
    Rectangle (333,118 80x32), "%s", text list: 'Sprachen', text index: 51
    Image (623,179 50x50), image: Icon.status_fehlerfrei_element
    Image (623,179 50x50), image: Icon.status_fehler_element
    Image (533,188 32x32), image: Icon.P_rechts
    Rectangle (433,188 80x32), "%s"
    Rectangle (333,188 80x32), "%s"
    Image (623,214 50x50), image: Icon.status_fehlerfrei_element
    Image (623,214 50x50), image: Icon.status_fehler_element
    Image (533,223 32x32), image: Icon.P_rechts
    Rectangle (433,223 80x32), "%s"
    Rectangle (333,223 80x32), "%s"
    Image (623,249 50x50), image: Icon.status_fehlerfrei_element
    Image (623,249 50x50), image: Icon.status_fehler_element
    Image (533,258 32x32), image: Icon.P_rechts
    Rectangle (433,258 80x32), "%s"
    Rectangle (333,258 80x32), "%s"
    Image (623,284 50x50), image: Icon.status_fehlerfrei_element
    Image (623,284 50x50), image: Icon.status_fehler_element
    Image (533,293 32x32), image: Icon.P_rechts
    Rectangle (433,293 80x32), "%s"
    Rectangle (333,293 80x32), "%s"
    Image (623,319 50x50), image: Icon.status_fehlerfrei_element
    Image (623,319 50x50), image: Icon.status_fehler_element
    Image (533,328 32x32), image: Icon.P_rechts
    Rectangle (433,328 80x32), "%s"
    Rectangle (333,328 80x32), "%s"
    Image (623,354 50x50), image: Icon.status_fehlerfrei_element
    Image (623,354 50x50), image: Icon.status_fehler_element
    Image (533,363 32x32), image: Icon.P_rechts
    Rectangle (433,363 80x32), "%s"
    Rectangle (333,363 80x32), "%s"
    Image (623,389 50x50), image: Icon.status_fehlerfrei_element
    Image (623,389 50x50), image: Icon.status_fehler_element
    Image (533,398 32x32), image: Icon.P_rechts
    Rectangle (433,398 80x32), "%s"
    Rectangle (333,398 80x32), "%s"
    Image (623,424 50x50), image: Icon.status_fehlerfrei_element
    Image (623,424 50x50), image: Icon.status_fehler_element
    Image (533,433 32x32), image: Icon.P_rechts
    Rectangle (433,433 80x32), "%s"
    Rectangle (333,433 80x32), "%s"
    Image (623,459 50x50), image: Icon.status_fehlerfrei_element
    Image (623,459 50x50), image: Icon.status_fehler_element
    Image (533,468 32x32), image: Icon.P_rechts
    Rectangle (433,468 80x32), "%s"
    Rectangle (333,468 80x32), "%s"
    Image (623,494 50x50), image: Icon.status_fehlerfrei_element
    Image (623,494 50x50), image: Icon.status_fehler_element
    Image (533,503 32x32), image: Icon.P_rechts
    Rectangle (433,503 80x32), "%s"
    Rectangle (333,503 80x32), "%s"
    Image (623,529 50x50), image: Icon.status_fehlerfrei_element
    Image (623,529 50x50), image: Icon.status_fehler_element
    Image (533,538 32x32), image: Icon.P_rechts
    Rectangle (433,538 80x32), "%s"
    Rectangle (333,538 80x32), "%s"
    Rectangle (0,0 800x50), "%s", text list: 'Sprachen', text index: 44
    Rectangle (0,55 128x58), "%s", text list: 'Sprachen', text index: 45
        OnMouseClick: execute { GWP_Library.Visu.i_Frame_Index:=0; }
    Rectangle (134,55 128x58), "%s", text list: 'Sprachen', text index: 46
        OnMouseClick: execute { GWP_Library.Visu.i_Frame_Index:=1; }
    Rectangle (268,55 128x58), "%s", text list: 'Sprachen', text index: 47
        OnMouseClick: execute { GWP_Library.Visu.i_Frame_Index:=2; }
    Rectangle (402,55 128x58), "%s", text list: 'Sprachen', text index: 48
        OnMouseClick: execute { GWP_Library.Visu.i_Frame_Index:=3; }
    Rectangle (0,55 128x5)
    Rectangle (134,55 128x5)
    Rectangle (268,55 128x5)
    Rectangle (402,55 128x5)
END_VISUALIZATION

// VISUs/IBN/Liste_AO
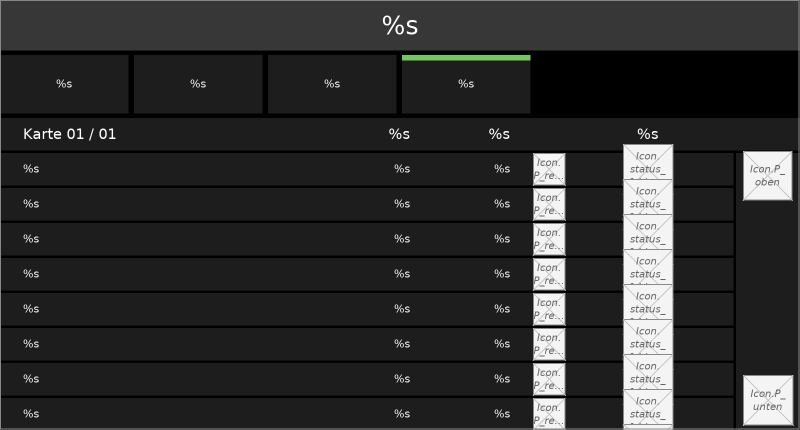
VISUALIZATION Liste_AO  // 800x430
    Rectangle (736,153 64x277)
    Image (743,375 50x50), image: Icon.P_unten
        OnMouseClick: execute {  }
    Image (743,151 49x49), image: Icon.P_oben
    Rectangle (0,153 733x32)
    Rectangle (20,153 400x32), "%s"
    Rectangle (0,223 733x32)
    Rectangle (20,223 400x32), "%s"
    Rectangle (0,188 733x32)
    Rectangle (20,188 400x32), "%s"
    Rectangle (0,258 733x32)
    Rectangle (20,258 400x32), "%s"
    Rectangle (0,328 733x32)
    Rectangle (20,328 400x32), "%s"
    Rectangle (0,293 733x32)
    Rectangle (20,293 400x32), "%s"
    Rectangle (0,538 733x32)
    Rectangle (20,538 400x32), "%s"
    Rectangle (0,363 733x32)
    Rectangle (20,363 400x32), "%s"
    Rectangle (0,433 733x32)
    Rectangle (20,433 400x32), "%s"
    Rectangle (0,398 733x32)
    Rectangle (20,398 400x32), "%s"
    Rectangle (0,468 733x32)
    Rectangle (20,468 400x32), "%s"
    Rectangle (0,503 733x32)
    Rectangle (20,503 400x32), "%s"
    Rectangle (0,118 800x32)
    Rectangle (20,118 324x32), "Karte 01 / 01"
    Rectangle (623,118 50x32), "%s", text list: 'Sprachen', text index: 49
    Image (623,144 50x50), image: Icon.status_fehlerfrei_element
    Image (623,144 50x50), image: Icon.status_fehler_element
    Image (533,153 32x32), image: Icon.P_rechts
        OnMouseClick: execute { GWP_Library.Visu.i_Frame_Index:=4; }
    Rectangle (433,153 80x32), "%s"
    Rectangle (333,153 80x32), "%s"
    Rectangle (433,118 80x32), "%s", text list: 'Sprachen', text index: 50
    Rectangle (333,118 80x32), "%s", text list: 'Sprachen', text index: 51
    Image (623,179 50x50), image: Icon.status_fehlerfrei_element
    Image (623,179 50x50), image: Icon.status_fehler_element
    Image (533,188 32x32), image: Icon.P_rechts
    Rectangle (433,188 80x32), "%s"
    Rectangle (333,188 80x32), "%s"
    Image (623,214 50x50), image: Icon.status_fehlerfrei_element
    Image (623,214 50x50), image: Icon.status_fehler_element
    Image (533,223 32x32), image: Icon.P_rechts
    Rectangle (433,223 80x32), "%s"
    Rectangle (333,223 80x32), "%s"
    Image (623,249 50x50), image: Icon.status_fehlerfrei_element
    Image (623,249 50x50), image: Icon.status_fehler_element
    Image (533,258 32x32), image: Icon.P_rechts
    Rectangle (433,258 80x32), "%s"
    Rectangle (333,258 80x32), "%s"
    Image (623,284 50x50), image: Icon.status_fehlerfrei_element
    Image (623,284 50x50), image: Icon.status_fehler_element
    Image (533,293 32x32), image: Icon.P_rechts
    Rectangle (433,293 80x32), "%s"
    Rectangle (333,293 80x32), "%s"
    Image (623,319 50x50), image: Icon.status_fehlerfrei_element
    Image (623,319 50x50), image: Icon.status_fehler_element
    Image (533,328 32x32), image: Icon.P_rechts
    Rectangle (433,328 80x32), "%s"
    Rectangle (333,328 80x32), "%s"
    Image (623,354 50x50), image: Icon.status_fehlerfrei_element
    Image (623,354 50x50), image: Icon.status_fehler_element
    Image (533,363 32x32), image: Icon.P_rechts
    Rectangle (433,363 80x32), "%s"
    Rectangle (333,363 80x32), "%s"
    Image (623,389 50x50), image: Icon.status_fehlerfrei_element
    Image (623,389 50x50), image: Icon.status_fehler_element
    Image (533,398 32x32), image: Icon.P_rechts
    Rectangle (433,398 80x32), "%s"
    Rectangle (333,398 80x32), "%s"
    Image (623,424 50x50), image: Icon.status_fehlerfrei_element
    Image (623,424 50x50), image: Icon.status_fehler_element
    Image (533,433 32x32), image: Icon.P_rechts
    Rectangle (433,433 80x32), "%s"
    Rectangle (333,433 80x32), "%s"
    Image (623,459 50x50), image: Icon.status_fehlerfrei_element
    Image (623,459 50x50), image: Icon.status_fehler_element
    Image (533,468 32x32), image: Icon.P_rechts
    Rectangle (433,468 80x32), "%s"
    Rectangle (333,468 80x32), "%s"
    Image (623,494 50x50), image: Icon.status_fehlerfrei_element
    Image (623,494 50x50), image: Icon.status_fehler_element
    Image (533,503 32x32), image: Icon.P_rechts
    Rectangle (433,503 80x32), "%s"
    Rectangle (333,503 80x32), "%s"
    Image (623,529 50x50), image: Icon.status_fehlerfrei_element
    Image (623,529 50x50), image: Icon.status_fehler_element
    Image (533,538 32x32), image: Icon.P_rechts
    Rectangle (433,538 80x32), "%s"
    Rectangle (333,538 80x32), "%s"
    Rectangle (0,0 800x50), "%s", text list: 'Sprachen', text index: 44
    Rectangle (0,55 128x58), "%s", text list: 'Sprachen', text index: 45
        OnMouseClick: execute { GWP_Library.Visu.i_Frame_Index:=0; }
    Rectangle (134,55 128x58), "%s", text list: 'Sprachen', text index: 46
        OnMouseClick: execute { GWP_Library.Visu.i_Frame_Index:=1; }
    Rectangle (268,55 128x58), "%s", text list: 'Sprachen', text index: 47
        OnMouseClick: execute { GWP_Library.Visu.i_Frame_Index:=2; }
    Rectangle (402,55 128x58), "%s", text list: 'Sprachen', text index: 48
        OnMouseClick: execute { GWP_Library.Visu.i_Frame_Index:=3; }
    Rectangle (0,55 128x5)
    Rectangle (134,55 128x5)
    Rectangle (268,55 128x5)
    Rectangle (402,55 128x5)
END_VISUALIZATION

// VISUs/IBN/Liste_DI
